(*

short summary
=================
This interface provides assert statements for 32 bit date and time ``DT``  

.. <legal notes>

legal notes
=================
| SPDX-FileCopyrightText: © 2022 ekvip automation GmbH <info@ekvip.de>
| SPDX-License-Identifier: Apache-2.0
| For details check: Apache-2.0_

.. _Apache-2.0: https://www.apache.org/licenses/LICENSE-2.0

.. </legal notes>

methods
==================

*)

INTERFACE I32BitDtAssertions EXTENDS __SYSTEM.IQueryInterface

(*

short summary
=================
This assertion method checks if the current value is equal to the expected value

.. <legal notes>

legal notes
=================
| SPDX-FileCopyrightText: © 2022 ekvip automation GmbH <info@ekvip.de>
| SPDX-License-Identifier: Apache-2.0
| For details check: Apache-2.0_

.. _Apache-2.0: https://www.apache.org/licenses/LICENSE-2.0

.. </legal notes>

parameters
=================

*)

METHOD valueIsEqualTo
VAR_INPUT
	(* current value to check *)
	currentValue	:DT;
	(* expected value to compare *)
	expectedValue	:DT;
	(* message if the assertion is false *)
	message			:AssertMessage;
END_VAR
END_METHOD

(*

short summary
=================
This assertion method checks if the current value is greater than the less value

.. <legal notes>

legal notes
=================
| SPDX-FileCopyrightText: © 2022 ekvip automation GmbH <info@ekvip.de>
| SPDX-License-Identifier: Apache-2.0
| For details check: Apache-2.0_

.. _Apache-2.0: https://www.apache.org/licenses/LICENSE-2.0

.. </legal notes>

parameters
=================

*)

METHOD valueIsGreaterThan
VAR_INPUT
	(* current value to check *)
	currentValue	:DT;
	(* less than lower limit *)
	lessValue		:DT;
	(* message if the assertion is false *)
	message			:AssertMessage;
END_VAR
END_METHOD

(*

short summary
=================
This assertion method checks if the current value is inside a limit

.. attention:: 
	limits are included: ``valueIsInRangeOf(dt#1970-01-01-0:0:0, dt#1970-01-01-0:0:0, dt#1970-01-01-0:0:0)``
	is a true assertion

.. <legal notes>

legal notes
=================
| SPDX-FileCopyrightText: © 2022 ekvip automation GmbH <info@ekvip.de>
| SPDX-License-Identifier: Apache-2.0
| For details check: Apache-2.0_

.. _Apache-2.0: https://www.apache.org/licenses/LICENSE-2.0

.. </legal notes>

parameters
=================

*)

METHOD valueIsInRangeOf
VAR_INPUT
	(* lower limit for the current value *)
	lowerLimit		:DT;
	(* current value to check *)
	currentValue	:DT;
	(* upper limit for the current value *)
	upperLimit		:DT;
	(* message if the assertion is false *)
	message			:AssertMessage;
END_VAR
END_METHOD

(*

short summary
=================
This assertion method checks if the current value is less than the greater value

.. <legal notes>

legal notes
=================
| SPDX-FileCopyrightText: © 2022 ekvip automation GmbH <info@ekvip.de>
| SPDX-License-Identifier: Apache-2.0
| For details check: Apache-2.0_

.. _Apache-2.0: https://www.apache.org/licenses/LICENSE-2.0

.. </legal notes>

parameters
=================

*)

METHOD valueIsLessThan
VAR_INPUT
	(* current value to check *)
	currentValue	:DT;
	(* greater than upper limit *)
	greaterValue	:DT;
	(* message if the assertion is false *)
	message			:AssertMessage;
END_VAR
END_METHOD

(*

short summary
=================
This assertion method checks if the current value is less than or equal to the maximum value

.. <legal notes>

legal notes
=================
| SPDX-FileCopyrightText: © 2022 ekvip automation GmbH <info@ekvip.de>
| SPDX-License-Identifier: Apache-2.0
| For details check: Apache-2.0_

.. _Apache-2.0: https://www.apache.org/licenses/LICENSE-2.0

.. </legal notes>

parameters
=================

*)

METHOD valueIsMax
VAR_INPUT
	(* current value to check *)
	currentValue	:DT;
	(* upper limit for the current value *)
	maximumValue	:DT;
	(* message if the assertion is false *)
	message			:AssertMessage;
END_VAR
END_METHOD

(*

short summary
=================
This assertion method checks if the current value is greater than or equal to the minimum value

.. <legal notes>

legal notes
=================
| SPDX-FileCopyrightText: © 2022 ekvip automation GmbH <info@ekvip.de>
| SPDX-License-Identifier: Apache-2.0
| For details check: Apache-2.0_

.. _Apache-2.0: https://www.apache.org/licenses/LICENSE-2.0

.. </legal notes>

parameters
=================

*)

METHOD valueIsMin
VAR_INPUT
	(* current value to check *)
	currentValue	:DT;
	(* lower limit for the current value *)
	minimumValue	:DT;
	(* message if the assertion is false *)
	message			:AssertMessage;
END_VAR
END_METHOD

(*

short summary
=================
This assertion method checks if the current value is not equal to the unexpected value

.. <legal notes>

legal notes
=================
| SPDX-FileCopyrightText: © 2022 ekvip automation GmbH <info@ekvip.de>
| SPDX-License-Identifier: Apache-2.0
| For details check: Apache-2.0_

.. _Apache-2.0: https://www.apache.org/licenses/LICENSE-2.0

.. </legal notes>

parameters
=================

*)

METHOD valueIsNotEqualTo
VAR_INPUT
	(* current value to check *)
	currentValue	:DT;
	(* unexpected value to compare *)
	unexpectedValue	:DT;
	(* message if the assertion is false *)
	message			:AssertMessage;
END_VAR
END_METHOD

END_INTERFACE

(* stored: Version 1.1.0.1, ProductVersion 3.1.4026.8
   Itf I32BitDtAssertions: Id {5a905069-b227-4488-ab1b-35ecbf038aaa}
   Method valueIsEqualTo: Id {6a1375d1-e0d9-48e1-86cc-c30e94f82508}
   Method valueIsGreaterThan: Id {af176cdc-55f1-428b-9f49-ef69f65f8946}
   Method valueIsInRangeOf: Id {0b20b21b-e5e3-4b99-8f78-333782f7590f}
   Method valueIsLessThan: Id {538cf9a5-5c49-4c7b-ad0b-b7c8fedfc9b4}
   Method valueIsMax: Id {6a43b931-5c6f-41ce-a5d0-54d4e23242f6}
   Method valueIsMin: Id {77b4b420-800f-4423-9122-05c68a088f7a}
   Method valueIsNotEqualTo: Id {166b488a-51d4-4561-bc99-d84b01853e17} *)
